// TIA Portal V17 export
// export: Created 2023-02-13T11:16:44.6337193Z, ExportSetting WithDefaults, DisplayName Totally Integrated Automation Portal, DisplayVersion V17, DisplayName TIA Portal Openness, DisplayVersion V17, DisplayName TIA Portal Teamcenter Gateway, DisplayVersion V17, DisplayName TIA Portal Version Control Interface, DisplayVersion V17, DisplayName SINAMICS Startdrive Advanced, DisplayVersion V17, DisplayName SINAMICS Startdrive G130, G150, S120, S150, SINAMICS MV, S210, DisplayVersion V17, DisplayName SINAMICS Startdrive G110M, G120, G120C, G120D, G120P, G115D, DisplayVersion V17, DisplayName STEP 7 Professional, DisplayVersion V17, DisplayName STEP 7 Safety, DisplayVersion V17, DisplayName WinCC Professional, DisplayVersion V17
DATA_BLOCK "Gen_Storage"   // DB15
{ S7_Optimized_Access := 'TRUE' }
VERSION : 0.1
// stored: AutoNumber false, DBAccessibleFromOPCUA true, DBAccessibleFromWebserver true, IsOnlyStoredInLoadMemory false, IsRetainMemResEnabled false, IsWriteProtectedInAS false, MemoryReserve 100
   VAR
      "Timer" : Struct
         Off_DrainIn_23 : TOF_TIME;
         Off_DrainIn_24_1 { S7_SetPoint := 'True'} : TOF_TIME;
         Off_DrainIn_24_2 { S7_SetPoint := 'True'} : TOF_TIME;
         Off_DrainIn_33 { S7_SetPoint := 'True'} : TOF_TIME;
         Off_DrainIn_34 { S7_SetPoint := 'True'} : TOF_TIME;
         Off_DrainIn_35 { S7_SetPoint := 'True'} : TOF_TIME;
         Off_DrainIn_79_1 { S7_SetPoint := 'True'} : TOF_TIME;
         Off_DrainIn_79_2 { S7_SetPoint := 'True'} : TOF_TIME;
         Off_DrainIn_79_3 { S7_SetPoint := 'True'} : TOF_TIME;
         Off_DrainIn_81 { S7_SetPoint := 'True'} : TOF_TIME;
         Off_DrainIn_84 { S7_SetPoint := 'True'} : TOF_TIME;
         Off_DrainIn_85 { S7_SetPoint := 'True'} : TOF_TIME;
      END_STRUCT;
      "THE4 CIP" : Struct
         "CIP Enable" : Bool;
         "CIP Request" : Bool;
         "CIP Line OK" : Bool;
         "CIP on Prog" : Bool;
         V_CIP_Cmd : Bool;
         p_trig : Bool;
      END_STRUCT;
      "THE5 CIP" : Struct
         "CIP Enable" : Bool;
         "CIP Request" : Bool;
         "CIP Line OK" : Bool;
         "CIP on Prog" : Bool;
         V_CIP_Cmd : Bool;
         p_trig : Bool;
      END_STRUCT;
   END_VAR
BEGIN
   "Timer".Off_DrainIn_23.PT := T#3s;
   "Timer".Off_DrainIn_24_1.PT := T#3s;
   "Timer".Off_DrainIn_33.PT := T#3s;
   "Timer".Off_DrainIn_34.PT := T#3s;
   "Timer".Off_DrainIn_35.PT := T#3s;
   "Timer".Off_DrainIn_79_1.PT := T#3s;
   "Timer".Off_DrainIn_81.PT := T#3s;
   "Timer".Off_DrainIn_84.PT := T#3s;
   "Timer".Off_DrainIn_85.PT := T#3s;
END_DATA_BLOCK
